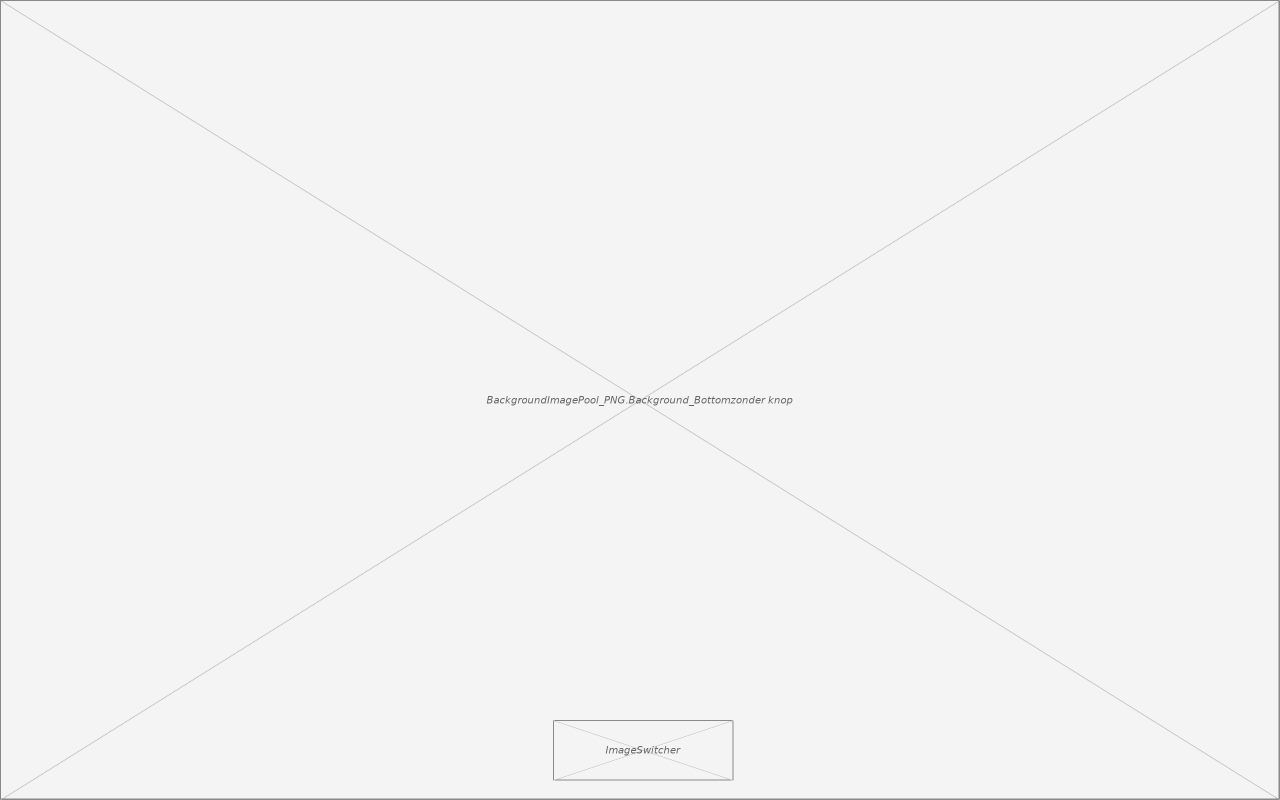
VISUALIZATION Background_SafetyAndSettings_SVG  // 1280x800
VAR_INPUT
	bHideEstop 			: BOOL ; // Hide emergency stop screen
	bDisableSettings	: BOOL ; // Deactivate settings
END_VAR
VAR_IN_OUT
	bCmdSettings	: BOOL ; // go to settings screen command
END_VAR
    Image (0,0 1280x800), invisible if: bHideEstop, input disabled if: bHideEstop, image: BackGroundImagePool_SVG.Emergency Stop Active 1280 x 800 Red Filled
    Image (0,0 1280x800), image: BackgroundImagePool_PNG.Background_Bottomzonder knop
    ImageSwitcher (553,720 180x60), variable: GVL_HMI.bCmdSettings, input disabled if: bDisableSettings, background image: Buttons_PNG.Home-Settings Switch Pushed, image: Buttons_PNG.Home-Settings Switch, behaviour: TOGGLE
        p3148411668: Buttons_PNG.Home-Settings Switch Pushed
END_VISUALIZATION

(* stored: Version 1.1.0.1, ProductVersion 3.1.4024.11
   Visu Background_SafetyAndSettings_SVG: Id {c9ed7bcb-f574-4619-a734-3f41a3d9ee6f} *)
